FUNCTION FC_SQL_InsertCommands : STRING(255)
VAR_INPUT
    iSensorValue: INT;
    iSampleNr: INT;
END_VAR

FC_SQL_InsertCommands := 'INSERT INTO [db_accessadmin].[TempSensor_Data] (SensorValue, SampleNr, Time) VALUES (';
FC_SQL_InsertCommands := CONCAT(FC_SQL_InsertCommands, INT_TO_STRING(iSensorValue));
FC_SQL_InsertCommands := CONCAT(FC_SQL_InsertCommands, ', ');
FC_SQL_InsertCommands := CONCAT(FC_SQL_InsertCommands, INT_TO_STRING(iSampleNr));
FC_SQL_InsertCommands := CONCAT(FC_SQL_InsertCommands, ', GETDATE());');

END_FUNCTION

(* stored: Version 1.1.0.1
   POU FC_SQL_InsertCommands: Id {d2e125de-b9e6-4fa0-b63a-88b16c7e6828}, SpecialFunc None *)
